// TIA Portal V20 export
// export: Created 2025-12-01T14:56:22.2508051Z, ExportSetting None, DisplayName Totally Integrated Automation Portal, DisplayVersion V20 Update 3, DisplayName TIA Portal Openness, DisplayVersion V20 Update 3, DisplayName TIA Portal Version Control Interface, DisplayVersion V20 Update 3, DisplayName STEP 7 Professional, DisplayVersion V20 Update 3, DisplayName STEP 7 Safety, DisplayVersion V20 Update 2, DisplayName WinCC Basic/Comfort/Advanced, DisplayVersion V20 Update 3, DisplayName WinCC Professional, DisplayVersion V20 Update 3, DisplayName WinCC Unified, DisplayVersion V20 Update 3
TYPE "NDD_HMI"
   STRUCT
      Entradas : Struct
         Byte_0_1 : Struct
            Libre_00 : Bool;
            S_NDD_ON : Bool;
            S_NDD_RE : Bool;
            Libre_003 : Bool;
            S_NDD_AUT : Bool;
            S_NDD_OFF : Bool;
            S_NDD_AV1 : Bool;   // Selector Cota 0m (ARMARIO)
            S_NDD_RET1 : Bool;   // Selector Cota 0m (ARMARIO)
            S_NDD_SE1 : Bool;   // Preselector Cota 0m (ARMARIO)
            S_NDD_SE2 : Bool;   // Preselector Cota 0m (ARMARIO)
            S_NDD_SE3 : Bool;   // Preselector Cota 0m (ARMARIO)
            S_NDD_SE4 : Bool;   // Preselector Cota 0m (ARMARIO)
            S_NDD_SE5 : Bool;   // Preselector Cota paletizado
            S_NDD_SE6 : Bool;   // Preselector Cota paletizado
            S_NDD_SE7 : Bool;   // Preselector Cota paletizado
            S_NDD_SE8 : Bool;   // Preselector Cota paletizado
         END_STRUCT;
         Byte_2_3 : Struct
            S_NDD_UP : Bool;   // Pulsador de Subir Elevador en el Puesto
            S_NDD_DW : Bool;   // Pulsador de Bajar Elevador en el Puesto
            S_NDD_CRG : Bool;   // Pulsador de Bajar Capa en el Puesto
            Libre_003 : Bool;
            Libre_004 : Bool;
            B_NDD_BARCajonera : Bool;   // Barrera Cajonera, debajo de Uñas --> Anulado ??
            S_NDD_AV2 : Bool;   // Selector Cota paletizado
            S_NDD_RET2 : Bool;   // Selector Cota paletizado
            QBE_NDD : Bool;   // Termico freno Elevacion
            QB_TElevador : Bool;   // Termico freno Transportador del Elevador --> En Variador
            B_TElevador_SEG : Bool;   // Sensor Posicionamiento OK
            B_TElevador_VEL : Bool;   // Sensor Corte Velocidad
            B_TElevador_1 : Bool;   // Sensor Parada
            Libre_015 : Bool;
            K_Enfardadora_PERM : Bool;   // Permiso Movimineto Manual Enfardadora (Elvador OK) Interlock
            Q_Enfardadora : Bool;   // Termico Enfardadora
         END_STRUCT;
         Byte_4_5 : Struct
            BF_NDD_BULSEG1 : Bool;   // Micro Mastil 1 (Bulon)
            BF_NDD_BULSEG2 : Bool;   // Micro Mastil 2 (Bulon)
            Libre_002 : Bool;
            LIbre_003 : Bool;
            S_BAREntrada_RE : Bool;   // Boton Rearme Muting Entrada
            S_BARSalida_RE : Bool;   // Boton Rearme Muting Salida
            S_MEEntrada_SUB : Bool;   // Boton SUBIR Mesa Elevadora Entrada
            S_MESalida_SUB : Bool;   // Boton SUBIR Mesa Elevadora Salida
            QB_TEntrada : Bool;   // Termico Freno Transportador Entrada --> En Variador
            B_TEntrada_1 : Bool;   // Sensor Parada Transportador Entrada
            B_TEntrada_PR1 : Bool;   // Sensor Protusion Transportadora Entrada (inicio)
            B_TEntrada_PR2 : Bool;   // Sensor Protusion Transportador Entrada (fin)
            B_MEEntrada_BMP : Bool;   // Sensor Bumper Contorno Mesa Elevadora Entrada
            QE_MEEntrada : Bool;   // Termico Elevación Mesa Elevadora Entrada
            B_MEEntrada_UP : Bool;   // Detector Arriba Mesa Elevadora Entrada
            B_MEEntrada_DW : Bool;   // Detector Abajo Mesa Elevadora Entrada
         END_STRUCT;
         Byte_6_7 : Struct
            QB_TSalida : Bool;   // Termico freno Transportador Salida --> En Variador
            B_TSalida_1 : Bool;   // Sensor Parada Transportadora Salida
            B_TSalida_PR1 : Bool;   // Sensor Protusion Transportador Salida entrada ---> En Entradas Seguras
            B_TSalida_PR2 : Bool;   // Sensor Protusion Transportador Salida
            B_MESalida_BMP : Bool;   // Sensor Bumper Contorno Mesa Elevadora Salida
            QE_MESalida : Bool;   // Termico Elevación Mesa Elevadora Salida
            B_MESalida_UP : Bool;   // Detector Arriba Mesa Elevadora Salida ---> En Entradas Seguras
            B_MESalida_DW : Bool;   // Detector Abajo Mesa Elevadora Salida ---> En Entradas Seguras
            KE_NDD_STOOK : Bool;   // STO Elevador
            K_TEelavador_STOOK : Bool;   // STO Transp. Elevador
            K_TSalida_STOOK : Bool;   // STO Transp. Anterior Posterior a Elevador
            K_TEntrada_STOOK : Bool;   // STO Transp. Posterior Anterior a Elevador
            KE_ME_STOOK : Bool;   // "STO" Elevacion Mesas Elevadoras
            K_Horquilla_STOOK : Bool;   // STO Horquilla
            K_Garra_STOOK : Bool;   // STO Uñas
            K_Enfardora_POTOK : Bool;   // Confirmación Enfardadora
         END_STRUCT;
         Byte_8_9 : Struct
            B_NDD_DIM1 : Bool;   // Control de Dimensiones para el Hueco
            B_NDD_DIM2 : Bool;   // Control de Dimensiones para el Hueco
            B_NDD_DIM3 : Bool;   // Control de Dimensiones para el Hueco
            B_NDD_DIM4 : Bool;   // Control de Dimensiones para el Hueco
            B_NDD_CRG1 : Bool;   // barrera control carga 1
            B_NDD_CRG2 : Bool;   // barrera control carga 2
            B_NDD_CRG3 : Bool;   // barrera control carga 3
            B_NDD_CRG4 : Bool;   // barrera control carga 4
            B_Horquilla_1 : Bool;   // Presencia palet en Horquilla
            B_Horquilla_PR1 : Bool;   // Protusion Horquilla
            Libre_012 : Bool;
            BF_Horquilla_OU : Bool;   // Limite pos horquilla retrocedido
            BF_Horquilla_IN : Bool;   // Limite pos horquilla avanzada
            B_Horquilla_IN : Bool;   // Posicion Horquilla avanzada
            QB_Horquilla : Bool;   // Termico freno Horquilla
            QB_Garra : Bool;   // Termico freno Uñas
         END_STRUCT;
         Byte_10_11 : Struct
            BF_Horquilla_UP1 : Bool;   // Sensor 1 proteccion horquilla Arriba
            BF_Horquilla_UP2 : Bool;   // Sensor 2 proteccion horquilla Arriba
            BF_Horquilla_UP3 : Bool;   // Sensor 3 proteccion horquilla Arriba
            BF_Horquilla_UP4 : Bool;   // Sensor 4 proteccion horquilla Arriba
            BF_Horquilla_DW1 : Bool;   // Sensor 1 proteccion horquilla Abajo
            BF_Horquilla_DW2 : Bool;   // Sensor 2 proteccion horquilla Abajo
            BF_Horquilla_DW3 : Bool;   // Sensor 3 proteccion horquilla Abajo
            BF_Horquilla_DW4 : Bool;   // Sensor 4 proteccion horquilla Abajo
            B_Garra_UP11 : Bool;   // Limite Uñas IZQ Arriba 1
            B_Garra_UP12 : Bool;   // Limite Uñas IZQ Arriba 2
            B_Garra_UP21 : Bool;   // Limite Uñas DER Arriba 1
            B_Garra_UP22 : Bool;   // Limite Uñas DER Arriba 2
            B_Garra_AL21 : Bool;   // Posicion Inicio Paletizado en Uñas Altura IZQ
            B_Garra_AL22 : Bool;   // Posicion Inicio Paletizado en Uñas Altura DER
            B_Garra_AL31 : Bool;   // Posicion Fin Paletizado en Uñas Altura IZQ
            B_Garra_AL32 : Bool;   // Posicion Fin Paletizado en Uñas Altura IZQ
         END_STRUCT;
         Byte_12_13 : Struct
            B_Garra_AL41_Escondida : Bool;   // Posicion unñas escondidas IZQ 1
            B_Garra_AL42_Escondida : Bool;   // Posicion unñas escondidas IZQ 2
            B_Garra_AL43_Escondida : Bool;   // Posicion unñas escondidas DER 1
            B_Garra_AL44_Escondida : Bool;   // Posicion unñas escondidas DER 1
            BF_Garra_DW11 : Bool;   // Limite Uñas IZQ Abajo 1
            BF_Garra_DW12 : Bool;   // Limite Uñas IZQ Abajo 2
            BF_Garra_DW21 : Bool;   // Limite Uñas DER Abajo 1
            BF_Garra_DW22 : Bool;   // Limite Uñas DER Abajo 2
            B_BAREntrada_MUT11 : Bool;   // Sensor 1 Muting entrada
            B_BAREntrada_MUT12 : Bool;   // Sensor 2 Muting entrada
            B_BAREntrada_MUT21 : Bool;   // Sensor 3 Muting entrada
            B_BAREntrada_MUT22 : Bool;   // Sensor 4 Muting entrada
            B_BARSalida_MUT11 : Bool;   // Sensor 1 Muting salida
            B_BARSalida_MUT12 : Bool;   // Sensor 2 Muting salida
            B_BARSalida_MUT21 : Bool;   // Sensor 3 Muting salida
            B_BARSalida_MUT22 : Bool;   // Sensor 4 Muting salida
         END_STRUCT;
      END_STRUCT;
      Salidas : Struct
         Byte_1_2 : Struct
            H_NDD_ON : Bool;   // Baliza Verde
            H_NDD_ER : Bool;   // Baliza Naranja
            H_NDD_ER2 : Bool;   // Baliza Roja
            H_NDD_RE : Bool;   // Piloto Rearme
            LIbre_004 : Bool;
            Libre_005 : Bool;
            Libre_006 : Bool;
            Libre_007 : Bool;
            H_NDD_ON_PU : Bool;   // Baliza Verde Puesto Operario
            H_NDD_ER_PU : Bool;   // Baliza Naranja Puesto Operario
            H_NDD_ER2_PU : Bool;   // Baliza Roja Puesto Operario
            H_NDD_AZU_PU : Bool;   // Baliza Azul Puesto Operario
            Libre_014 : Bool;
            Libre_015 : Bool;
            H_BAREntrada_MUT : Bool;   // Baliza Muting entrada
            H_BARSalida_MUT : Bool;   // Baliza Muting salida
         END_STRUCT;
         Byte_3_4 : Struct
            KMS_MEEntrada : Bool;   // Subir Mesa Elevadora Entrada
            KMB_MEEntrada : Bool;   // Bajar Mesa Elevadora Entrada
            KMS_MESalida : Bool;   // Subir Mesa Elevadora Salida
            KMB_MESalida : Bool;   // Bajar Mesa ElevadoraSalida
            Libre_004 : Bool;
            Libre_005 : Bool;
            Libre_006 : Bool;
            K_Enfardadora_MVOK : Bool;   // Elevador OK para Mover enfardadora (Interlock ENFARDADORA)
            Libre_010 : Bool;
            Libre_011 : Bool;
            Libre_012 : Bool;
            Libre_013 : Bool;
            Libre_014 : Bool;
            Libre_015 : Bool;
            Libre_016 : Bool;
            Libre_017 : Bool;
         END_STRUCT;
      END_STRUCT;
      EntradasSeguras : Struct
         Tarjeta_1 : Struct
            SF_NDD_EM : Bool;   // Seta Amarilla
            SF_NDD_UP : Bool;   // Micro del Elevador Arriba
            SF_NDD_DW : Bool;   // Micro del Elevador Abajo
            SF_NDD_BARPuesto : Bool;   // Barrera de Nivel de carga en el Puesto Paletizado
            Reservado_04 : Bool;
            Reservado_05 : Bool;
            Reservado_06 : Bool;
            Reservado_07 : Bool;
            Reservado_10 : Bool;
            Reservado_11 : Bool;
            Reservado_12 : Bool;
            Reservado_13 : Bool;
            Reservado_14 : Bool;
            Reservado_15 : Bool;
            Reservado_16 : Bool;
            Reservado_17 : Bool;
            Reservado_20 : Bool;
            Reservado_21 : Bool;
            Reservado_22 : Bool;
            Reservado_23 : Bool;
            Reservado_24 : Bool;
            Reservado_25 : Bool;
            Reservado_26 : Bool;
            Reservado_27 : Bool;
            Reservado_30 : Bool;
            Reservado_31 : Bool;
            Reservado_32 : Bool;
            Reservado_33 : Bool;
            Reservado_34 : Bool;
            Reservado_35 : Bool;
            Reservado_36 : Bool;
            Reservado_37 : Bool;
            Reservado_40 : Bool;
            Reservado_41 : Bool;
            Reservado_42 : Bool;
            Reservado_43 : Bool;
            Reservado_44 : Bool;
            Reservado_45 : Bool;
            Reservado_46 : Bool;
            Reservado_47 : Bool;
            Reservado_50 : Bool;
            Reservado_51 : Bool;
            Reservado_52 : Bool;
            Reservado_53 : Bool;
            Reservado_54 : Bool;
            Reservado_55 : Bool;
            Reservado_56 : Bool;
            Reservado_57 : Bool;
         END_STRUCT;
         Tarjeta_2 : Struct
            BF_NDD_CHEC1 : Bool;   // Elevador en Mesas Elevadoras
            BF_NDD_CHEC2 : Bool;   // Elevador en Cota Horquilla
            BF_NDD_CHEC3 : Bool;   // Elevador en Cota Uñas
            BF_NDD_CHEC4 : Bool;   // Elevador en Cota Enfardado
            Reservado_04 : Bool;
            Reservado_05 : Bool;
            Reservado_06 : Bool;
            Reservado_07 : Bool;
            Reservado_10 : Bool;
            Reservado_11 : Bool;
            Reservado_12 : Bool;
            Reservado_13 : Bool;
            Reservado_14 : Bool;
            Reservado_15 : Bool;
            Reservado_16 : Bool;
            Reservado_17 : Bool;
            Reservado_20 : Bool;
            Reservado_21 : Bool;
            Reservado_22 : Bool;
            Reservado_23 : Bool;
            Reservado_24 : Bool;
            Reservado_25 : Bool;
            Reservado_26 : Bool;
            Reservado_27 : Bool;
            Reservado_30 : Bool;
            Reservado_31 : Bool;
            Reservado_32 : Bool;
            Reservado_33 : Bool;
            Reservado_34 : Bool;
            Reservado_35 : Bool;
            Reservado_36 : Bool;
            Reservado_37 : Bool;
            Reservado_40 : Bool;
            Reservado_41 : Bool;
            Reservado_42 : Bool;
            Reservado_43 : Bool;
            Reservado_44 : Bool;
            Reservado_45 : Bool;
            Reservado_46 : Bool;
            Reservado_47 : Bool;
            Reservado_50 : Bool;
            Reservado_51 : Bool;
            Reservado_52 : Bool;
            Reservado_53 : Bool;
            Reservado_54 : Bool;
            Reservado_55 : Bool;
            Reservado_56 : Bool;
            Reservado_57 : Bool;
         END_STRUCT;
         Tarjeta_3 : Struct
            BF_MESalida_UP : Bool;   // Mesa Elevadora Salida UP
            BF_MESalida_DW : Bool;   // Mesa Elevadora Salida DW
            BF_BAREntrada_BAR1 : Bool;   // Barrera de Seguridad mesa de entrada
            BF_BARSalida_BAR1 : Bool;   // Barrera de Seguridad mesa de salida
            Reservado_04 : Bool;
            Reservado_05 : Bool;
            Reservado_06 : Bool;
            Reservado_07 : Bool;
            Reservado_10 : Bool;
            Reservado_11 : Bool;
            Reservado_12 : Bool;
            Reservado_13 : Bool;
            Reservado_14 : Bool;
            Reservado_15 : Bool;
            Reservado_16 : Bool;
            Reservado_17 : Bool;
            Reservado_20 : Bool;
            Reservado_21 : Bool;
            Reservado_22 : Bool;
            Reservado_23 : Bool;
            Reservado_24 : Bool;
            Reservado_25 : Bool;
            Reservado_26 : Bool;
            Reservado_27 : Bool;
            Reservado_30 : Bool;
            Reservado_31 : Bool;
            Reservado_32 : Bool;
            Reservado_33 : Bool;
            Reservado_34 : Bool;
            Reservado_35 : Bool;
            Reservado_36 : Bool;
            Reservado_37 : Bool;
            Reservado_40 : Bool;
            Reservado_41 : Bool;
            Reservado_42 : Bool;
            Reservado_43 : Bool;
            Reservado_44 : Bool;
            Reservado_45 : Bool;
            Reservado_46 : Bool;
            Reservado_47 : Bool;
            Reservado_50 : Bool;
            Reservado_51 : Bool;
            Reservado_52 : Bool;
            Reservado_53 : Bool;
            Reservado_54 : Bool;
            Reservado_55 : Bool;
            Reservado_56 : Bool;
            Reservado_57 : Bool;
         END_STRUCT;
         Tarjeta_4 : Struct
            SP_NDD_1 : Bool;   // Micro Puerta Cota 0
            SP_NDD_2 : Bool;   // Micro Puerta Pasarela Enfardadora (3,7)
            SP_NDD_3 : Bool;   // Micro Puerta Arriba cajonera horquilla
            "SCALING FACTOR" : Bool;   // SCALING FACTOR ELEVADOR
            Reservado_04 : Bool;
            Reservado_05 : Bool;
            Reservado_06 : Bool;
            Reservado_07 : Bool;
            Reservado_10 : Bool;
            Reservado_11 : Bool;
            Reservado_12 : Bool;
            Reservado_13 : Bool;
            Reservado_14 : Bool;
            Reservado_15 : Bool;
            Reservado_16 : Bool;
            Reservado_17 : Bool;
            Reservado_20 : Bool;
            Reservado_21 : Bool;
            Reservado_22 : Bool;
            Reservado_23 : Bool;
            Reservado_24 : Bool;
            Reservado_25 : Bool;
            Reservado_26 : Bool;
            Reservado_27 : Bool;
            Reservado_30 : Bool;
            Reservado_31 : Bool;
            Reservado_32 : Bool;
            Reservado_33 : Bool;
            Reservado_34 : Bool;
            Reservado_35 : Bool;
            Reservado_36 : Bool;
            Reservado_37 : Bool;
            Reservado_40 : Bool;
            Reservado_41 : Bool;
            Reservado_42 : Bool;
            Reservado_43 : Bool;
            Reservado_44 : Bool;
            Reservado_45 : Bool;
            Reservado_46 : Bool;
            Reservado_47 : Bool;
            Reservado_50 : Bool;
            Reservado_51 : Bool;
            Reservado_52 : Bool;
            Reservado_53 : Bool;
            Reservado_54 : Bool;
            Reservado_55 : Bool;
            Reservado_56 : Bool;
            Reservado_57 : Bool;
         END_STRUCT;
         Tarjeta_5 : Struct
            Libre_0 : Bool;
            Libre_1 : Bool;
            Libre_2 : Bool;
            Libre_3 : Bool;
            Reservado_04 : Bool;
            Reservado_05 : Bool;
            Reservado_06 : Bool;
            Reservado_07 : Bool;
            Reservado_10 : Bool;
            Reservado_11 : Bool;
            Reservado_12 : Bool;
            Reservado_13 : Bool;
            Reservado_14 : Bool;
            Reservado_15 : Bool;
            Reservado_16 : Bool;
            Reservado_17 : Bool;
            Reservado_20 : Bool;
            Reservado_21 : Bool;
            Reservado_22 : Bool;
            Reservado_23 : Bool;
            Reservado_24 : Bool;
            Reservado_25 : Bool;
            Reservado_26 : Bool;
            Reservado_27 : Bool;
            Reservado_30 : Bool;
            Reservado_31 : Bool;
            Reservado_32 : Bool;
            Reservado_33 : Bool;
            Reservado_34 : Bool;
            Reservado_35 : Bool;
            Reservado_36 : Bool;
            Reservado_37 : Bool;
            Reservado_40 : Bool;
            Reservado_41 : Bool;
            Reservado_42 : Bool;
            Reservado_43 : Bool;
            Reservado_44 : Bool;
            Reservado_45 : Bool;
            Reservado_46 : Bool;
            Reservado_47 : Bool;
            Reservado_50 : Bool;
            Reservado_51 : Bool;
            Reservado_52 : Bool;
            Reservado_53 : Bool;
            Reservado_54 : Bool;
            Reservado_55 : Bool;
            Reservado_56 : Bool;
            Reservado_57 : Bool;
         END_STRUCT;
         Tarjeta_6 : Struct
            SF_NDD_MAIN : Bool;   // Llave Mantenimiento
            SF_NDD_OFFL : Bool;   // Llave OFFLINE
            B_Horquilla_OU : Bool;   // Posicion Horquilla retrocedida
            B_TSalida_PR2 : Bool;   // Sensor Protusion Mesa Elevadora Salida
            Libre_4 : Bool;
            Libre_5 : Bool;
            Libre_6 : Bool;
            Libre_7 : Bool;
            Reservado_10 : Bool;
            Reservado_11 : Bool;
            Reservado_12 : Bool;
            Reservado_13 : Bool;
            Reservado_14 : Bool;
            Reservado_15 : Bool;
            Reservado_16 : Bool;
            Reservado_17 : Bool;
            Reservado_20 : Bool;
            Reservado_21 : Bool;
            Reservado_22 : Bool;
            Reservado_23 : Bool;
            Reservado_24 : Bool;
            Reservado_25 : Bool;
            Reservado_26 : Bool;
            Reservado_27 : Bool;
            Reservado_30 : Bool;
            Reservado_31 : Bool;
            Reservado_32 : Bool;
            Reservado_33 : Bool;
            Reservado_34 : Bool;
            Reservado_35 : Bool;
            Reservado_36 : Bool;
            Reservado_37 : Bool;
            Reservado_40 : Bool;
            Reservado_41 : Bool;
            Reservado_42 : Bool;
            Reservado_43 : Bool;
            Reservado_44 : Bool;
            Reservado_45 : Bool;
            Reservado_46 : Bool;
            Reservado_47 : Bool;
            Reservado_50 : Bool;
            Reservado_51 : Bool;
            Reservado_52 : Bool;
            Reservado_53 : Bool;
            Reservado_54 : Bool;
            Reservado_55 : Bool;
            Reservado_56 : Bool;
            Reservado_57 : Bool;
         END_STRUCT;
      END_STRUCT;
      SalidasSeguras : Struct
         Tarjeta_1 : Struct
            KFE_NDD_STO : Bool;   // STO Elevador
            KF_TElevador_STO : Bool;   // STO Transp. Elevador
            KF_TSalida_STO : Bool;   // STO Transp. Salida
            KF_TEntrada_STO : Bool;   // STO Transp. Entrada
            Reservado_04 : Bool;
            Reservado_05 : Bool;
            Reservado_06 : Bool;
            Reservado_07 : Bool;
            Reservado_10 : Bool;
            Reservado_11 : Bool;
            Reservado_12 : Bool;
            Reservado_13 : Bool;
            Reservado_14 : Bool;
            Reservado_15 : Bool;
            Reservado_16 : Bool;
            Reservado_17 : Bool;
            Reservado_20 : Bool;
            Reservado_21 : Bool;
            Reservado_22 : Bool;
            Reservado_23 : Bool;
            Reservado_24 : Bool;
            Reservado_25 : Bool;
            Reservado_26 : Bool;
            Reservado_27 : Bool;
            Reservado_30 : Bool;
            Reservado_31 : Bool;
            Reservado_32 : Bool;
            Reservado_33 : Bool;
            Reservado_34 : Bool;
            Reservado_35 : Bool;
            Reservado_36 : Bool;
            Reservado_37 : Bool;
            Reservado_40 : Bool;
            Reservado_41 : Bool;
            Reservado_42 : Bool;
            Reservado_43 : Bool;
            Reservado_44 : Bool;
            Reservado_45 : Bool;
            Reservado_46 : Bool;
            Reservado_47 : Bool;
            Reservado_50 : Bool;
            Reservado_51 : Bool;
            Reservado_52 : Bool;
            Reservado_53 : Bool;
            Reservado_54 : Bool;
            Reservado_55 : Bool;
            Reservado_56 : Bool;
            Reservado_57 : Bool;
         END_STRUCT;
         Tarjeta_2 : Struct
            KF_Horquillas_STO : Bool;   // STO Horquilla
            KF_Garras_STO : Bool;   // STO_Uñas
            KFP_NDD_BL1 : Bool;   // Desbloqueo puerta Cota 0 (elevador)
            KFE_ME_STO : Bool;   // "STO" Elevacion Mesas Elevadoras
            Reservado_04 : Bool;
            Reservado_05 : Bool;
            Reservado_06 : Bool;
            Reservado_07 : Bool;
            Reservado_10 : Bool;
            Reservado_11 : Bool;
            Reservado_12 : Bool;
            Reservado_13 : Bool;
            Reservado_14 : Bool;
            Reservado_15 : Bool;
            Reservado_16 : Bool;
            Reservado_17 : Bool;
            Reservado_20 : Bool;
            Reservado_21 : Bool;
            Reservado_22 : Bool;
            Reservado_23 : Bool;
            Reservado_24 : Bool;
            Reservado_25 : Bool;
            Reservado_26 : Bool;
            Reservado_27 : Bool;
            Reservado_30 : Bool;
            Reservado_31 : Bool;
            Reservado_32 : Bool;
            Reservado_33 : Bool;
            Reservado_34 : Bool;
            Reservado_35 : Bool;
            Reservado_36 : Bool;
            Reservado_37 : Bool;
            Reservado_40 : Bool;
            Reservado_41 : Bool;
            Reservado_42 : Bool;
            Reservado_43 : Bool;
            Reservado_44 : Bool;
            Reservado_45 : Bool;
            Reservado_46 : Bool;
            Reservado_47 : Bool;
            Reservado_50 : Bool;
            Reservado_51 : Bool;
            Reservado_52 : Bool;
            Reservado_53 : Bool;
            Reservado_54 : Bool;
            Reservado_55 : Bool;
            Reservado_56 : Bool;
            Reservado_57 : Bool;
         END_STRUCT;
         Tarjeta_3 : Struct
            KM_Enfardadora : Bool;   // Potencia Enfardadora
            KFP_Enfardadora_BL1 : Bool;   // Desbloqueo puerta Enfardadora
            Libre_2 : Bool;
            Libre_3 : Bool;
            Reservado_04 : Bool;
            Reservado_05 : Bool;
            Reservado_06 : Bool;
            Reservado_07 : Bool;
            Reservado_10 : Bool;
            Reservado_11 : Bool;
            Reservado_12 : Bool;
            Reservado_13 : Bool;
            Reservado_14 : Bool;
            Reservado_15 : Bool;
            Reservado_16 : Bool;
            Reservado_17 : Bool;
            Reservado_20 : Bool;
            Reservado_21 : Bool;
            Reservado_22 : Bool;
            Reservado_23 : Bool;
            Reservado_24 : Bool;
            Reservado_25 : Bool;
            Reservado_26 : Bool;
            Reservado_27 : Bool;
            Reservado_30 : Bool;
            Reservado_31 : Bool;
            Reservado_32 : Bool;
            Reservado_33 : Bool;
            Reservado_34 : Bool;
            Reservado_35 : Bool;
            Reservado_36 : Bool;
            Reservado_37 : Bool;
            Reservado_40 : Bool;
            Reservado_41 : Bool;
            Reservado_42 : Bool;
            Reservado_43 : Bool;
            Reservado_44 : Bool;
            Reservado_45 : Bool;
            Reservado_46 : Bool;
            Reservado_47 : Bool;
            Reservado_50 : Bool;
            Reservado_51 : Bool;
            Reservado_52 : Bool;
            Reservado_53 : Bool;
            Reservado_54 : Bool;
            Reservado_55 : Bool;
            Reservado_56 : Bool;
            Reservado_57 : Bool;
         END_STRUCT;
      END_STRUCT;
      Elevador : Struct
         ReferenciaOK : Bool;
         Libre_1 : Bool;
         Libre_2 : Bool;
         Libre_3 : Bool;
         Libre_4 : Bool;
         Libre_5 : Bool;
         Libre_6 : Bool;
         Libre_7 : Bool;
         PerEntrada_CotaME : Bool;
         PerEntrada_CotaEnfardado : Bool;
         PerEntrada_CotaPaletizado : Bool;
         Libre_13 : Bool;
         Libre_14 : Bool;
         Libre_15 : Bool;
         Libre_16 : Bool;
         Libre_17 : Bool;
         Posicion : Int;
      END_STRUCT;
      Horquilla : Struct
         ReferenciaOK : Bool;
         Libre_1 : Bool;
         Libre_2 : Bool;
         Libre_3 : Bool;
         Libre_4 : Bool;
         Libre_5 : Bool;
         Libre_6 : Bool;
         Libre_7 : Bool;
         Libre_10 : Bool;
         Libre_11 : Bool;
         Libre_12 : Bool;
         Libre_13 : Bool;
         Libre_14 : Bool;
         Libre_15 : Bool;
         Libre_16 : Bool;
         Libre_17 : Bool;
         Posicion : Int;
      END_STRUCT;
      Garra : Struct
         ReferenciaOK : Bool;
         Libre_1 : Bool;
         Libre_2 : Bool;
         Libre_3 : Bool;
         Libre_4 : Bool;
         Libre_5 : Bool;
         Libre_6 : Bool;
         Libre_7 : Bool;
         Libre_10 : Bool;
         Libre_11 : Bool;
         Libre_12 : Bool;
         Libre_13 : Bool;
         Libre_14 : Bool;
         Libre_15 : Bool;
         Libre_16 : Bool;
         Libre_17 : Bool;
         Posicion : Int;
      END_STRUCT;
   END_STRUCT;
END_TYPE
